// TIA Portal V17 export
// export: Created 2025-06-26T07:49:46.8777156Z, ExportSetting WithDefaults, DisplayName Totally Integrated Automation Portal, DisplayVersion V17 Update 8, DisplayName TIA Portal Openness, DisplayVersion V17 Update 8, DisplayName TIA Portal Version Control Interface, DisplayVersion V17, DisplayName STEP 7 Professional, DisplayVersion V17 Update 8, DisplayName STEP 7 Safety, DisplayVersion V17 Update 6, DisplayName WinCC Advanced, DisplayVersion V17 Update 8
FUNCTION_BLOCK "fbPI_Regulator"   // FB21, FBD
TITLE = PI Regulator
{ S7_Optimized_Access := 'TRUE' }
VERSION : 0.1
// stored: AutoNumber true, IsIECCheckEnabled false, IsRetainMemResEnabled false, MemoryReserve 0, SetENOAutomatically false, UDAEnableTagReadback false
   VAR_INPUT
      sPV : "stCalcValue";   // Process value
      fCycleTime : Real;
      bEnable : Bool;
      bReset : Bool;
   END_VAR
   VAR_OUTPUT
      fOut : Real;
      bAtMin : Bool;
      bAtMax : Bool;
   END_VAR
   VAR_IN_OUT
      sTag : "stPI_Regulator";
   END_VAR
   VAR
      D_Mem : Real;
      I_Mem : Real;
      Param_Mem : Real;
   END_VAR
   VAR_TEMP
      Enabled : Bool;
      fDeviation : Real;
   END_VAR
BEGIN

REGION Network 1: Reset manual mode
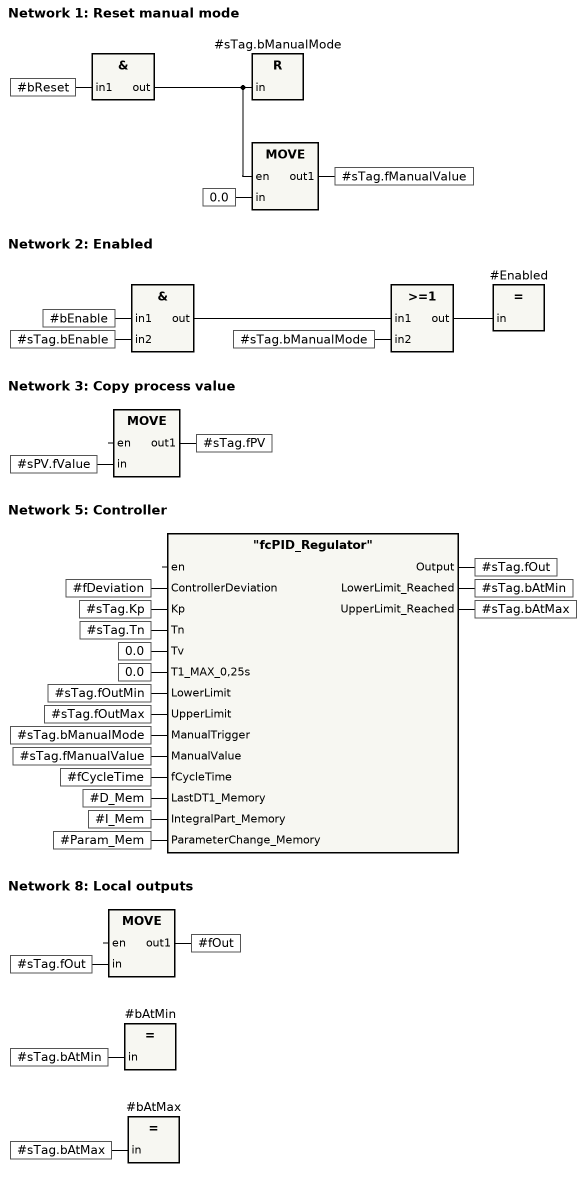
   IF #bReset THEN
       #sTag.bManualMode := FALSE;
       #sTag.fManualValue := 0.0;
   END_IF;
END_REGION

REGION Network 2: Enabled
   // Local input is from process control logic: when to run the regulator
   // Tag input is from HMI: do we want to run this regulator at all
   #Enabled := (#bEnable AND #sTag.bEnable) OR #sTag.bManualMode;
END_REGION

REGION Network 3: Copy process value
   #sTag.fPV := #sPV.fValue;
END_REGION

REGION Network 4 (SCL): Deviation
   // NaN detection
   IF "isNaN"(#sTag.fSP) OR "isNaN"(#sTag.fPV) THEN
       #fDeviation := 0.0;
       #sTag.bFault := TRUE;
   ELSE
       #fDeviation := #sTag.fSP - #sTag.fPV;
       #sTag.bFault := FALSE;
   END_IF;
END_REGION

REGION Network 5: Controller
   // NOTE: controller always runs regardless of mode
   "fcPID_Regulator"(ControllerDeviation := #fDeviation,
                     Kp := #sTag.Kp,
                     Tn := #sTag.Tn,
                     Tv := 0.0,
                     "T1_MAX_0,25s" := 0.0,
                     LowerLimit := #sTag.fOutMin,
                     UpperLimit := #sTag.fOutMax,
                     ManualTrigger := #sTag.bManualMode,
                     ManualValue := #sTag.fManualValue,
                     fCycleTime := #fCycleTime,
                     LastDT1_Memory := #D_Mem,
                     IntegralPart_Memory := #I_Mem,
                     ParameterChange_Memory := #Param_Mem,
                     Output => #sTag.fOut,
                     LowerLimit_Reached => #sTag.bAtMin,
                     UpperLimit_Reached => #sTag.bAtMax);
END_REGION

REGION Network 6 (SCL): Disable
   IF #Enabled = FALSE OR #sTag.bFault = TRUE THEN
       #sTag.fOut := 0.0;
       #sTag.bAtMin := FALSE;
       #sTag.bAtMax := FALSE;
   END_IF;
END_REGION

REGION Network 7 (SCL): Mode
   // Mode
   IF #sTag.bManualMode = TRUE THEN
       #sTag.nMode := 2;
   ELSIF #sTag.bEnable = TRUE THEN
       #sTag.nMode := 1;
   ELSE
       #sTag.nMode := 0;
   END_IF;
END_REGION

REGION Network 8: Local outputs
   #fOut := #sTag.fOut;
   #bAtMin := #sTag.bAtMin;
   #bAtMax := #sTag.bAtMax;
END_REGION
END_FUNCTION_BLOCK
